TYPE ST_System_SHZ_Parameter :
STRUCT
	Temp_Vorl_Max			: REAL	:= 65;
	Temp_Vorl_Min			: REAL	:= 30;

	Temp_Heisswasser_Max    : REAL;
	Temp_Heisswasser_Min    : REAL;

	Kennlinie_Heizung		: ST_Parameter_Kennlinie_Heizung_Kuehlung;
	Kennlinie_Tctr			: DINT := 5000;

	Nachtabsenkung_Mo		: ST_Parameter_Nachtabsenkung;
	Nachtabsenkung_Di		: ST_Parameter_Nachtabsenkung;
	Nachtabsenkung_Mi		: ST_Parameter_Nachtabsenkung;
	Nachtabsenkung_Do		: ST_Parameter_Nachtabsenkung;
	Nachtabsenkung_Fr		: ST_Parameter_Nachtabsenkung;
	Nachtabsenkung_Sa		: ST_Parameter_Nachtabsenkung;
	Nachtabsenkung_So		: ST_Parameter_Nachtabsenkung;

	AutoQuittierung			: BOOL := 0;
END_STRUCT
END_TYPE

(* stored: Version 1.1.0.1, ProductVersion 3.1.4024.9
   DUT ST_System_SHZ_Parameter: Id {67ee2a33-acd1-4af3-a0f2-c365b8864882} *)
